{attribute 'qualified_only'}
{attribute 'strict'}
{attribute 'to_string'}
TYPE E_SeqServo :
(
	IDLE := 0,
	STOP,
	RESET,
	HOME,
	HOME_SET_POSITION,
	HOME_READ_PARM,
	HOME_DISABLE_DRIVE,
	HOME_WRITE_PARM_PERS,
	HOME_ENABLE_DRIVE,
	JOG,
	MOVE_ABS,
	ERROR
);
END_TYPE

(* stored: Version 1.1.0.1, ProductVersion 3.1.4024.12
   DUT E_SeqServo: Id {af91c62d-b749-4f8b-b488-e5b765c287ff} *)
